PROGRAM MAIN
VAR
END_VAR

END_PROGRAM

(* stored: Version 1.1.0.1
   POU MAIN: Id {d8de5791-f153-470a-bfaa-453c619a7f06} *)
